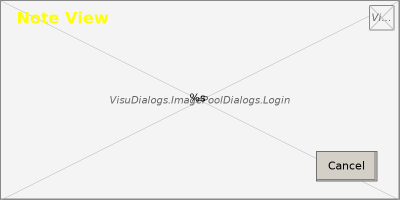
VISUALIZATION Note  // 400x200
VAR_IN_OUT
	noteHMI:NoteStruct;
END_VAR
    Image (0,0 400x200), image: VisuDialogs.ImagePoolDialogs.Login
    Rectangle (24,83 347x30), "%s", text variable: noteHMI.showText
    Button (316,151 61x30), "Cancel"
        OnMouseClick: execute { noteHMI.showFlag:=FALSE; }
    Image (369,5 25x25), image: VisuDialogs.ImagePoolDialogs.Delete
        OnMouseClick: execute { noteHMI.showFlag:=FALSE; }
    Label (5,3 116x30), "Note View"
END_VISUALIZATION

(* stored: Version 1.1.0.1, ProductVersion 3.1.4024.4
   Visu Note: Id {be73b368-8a44-4b11-9015-8d3170a20e50} *)
